Fanuc KAREL source: KB00113.KL

PROGRAM KB00113
%NOLOCKGROUP
%ENVIRONMENT KCLOP
VAR
  P1: STRING[80]
  P2: INTEGER
BEGIN
  P1 = 'A'
  P2 = 1
  KCL(P1, P2)
END KB00113
